FUNCTION_BLOCK FB_setupJnt5AdjustDetect
VAR_INPUT
END_VAR
VAR_OUTPUT
END_VAR
VAR
	m_pAutoAdjustOnCounts :INT :=0;
	m_nAutoAdjustOnCounts :INT :=0;
	m_adjustOnCountThres :INT :=50;
END_VAR

METHOD run : INT
VAR_INPUT
	IOValue :UDINT;
END_VAR

VAR_OUTPUT
	
END_VAR
// joint3 positive auto adjust is 3th bit
IF 2=(IOValue AND 10#2) THEN
	m_pAutoAdjustOnCounts :=MIN(m_pAutoAdjustOnCounts +1,m_adjustOnCountThres);
ELSE
	m_pAutoAdjustOnCounts :=0;
END_IF

// joint3 negative auto adjust is 2th bit
IF 1=(IOValue AND 10#1) THEN
	m_nAutoAdjustOnCounts :=MIN(m_nAutoAdjustOnCounts +1,m_adjustOnCountThres);
ELSE
	m_nAutoAdjustOnCounts :=0;
END_IF

IF m_pAutoAdjustOnCounts >= m_adjustOnCountThres THEN
	run :=1;
ELSIF m_nAutoAdjustOnCounts >= m_adjustOnCountThres THEN
	run := -1;
ELSE 
	run :=0;
END_IF
END_METHOD

END_FUNCTION_BLOCK

(* stored: Version 1.1.0.1, ProductVersion 3.1.4024.11
   POU FB_setupJnt5AdjustDetect: Id {11a489ef-1382-4370-ad13-f9936b9d700b}, SpecialFunc None
   Method run: Id {06d8fba5-ed28-4dd9-8f06-03d85a099ac5} *)
